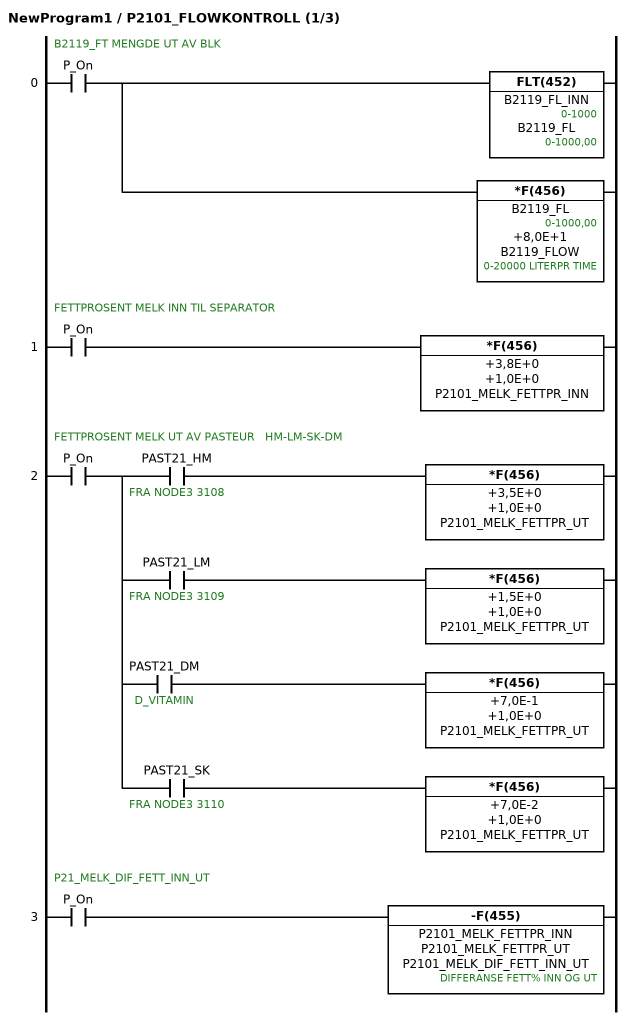
; [picture p1056: NewProgram1 / P2101_FLOWKONTROLL, rungs 0-3]
; rung 0: B2119_FT MENGDE UT AV BLK
LD P_On
FLT(452) B2119_FL_INN B2119_FL  ; 0-1000, 0-1000,00
*F(456) B2119_FL +8,0E+1 B2119_FLOW  ; 0-1000,00, 0-20000 LITERPR TIME
; rung 1: FETTPROSENT MELK INN TIL SEPARATOR
LD P_On
*F(456) +3,8E+0 +1,0E+0 P2101_MELK_FETTPR_INN
; rung 2: FETTPROSENT MELK UT AV PASTEUR   HM-LM-SK-DM
LD P_On
OUT TR0
AND PAST21_HM  ; FRA NODE3 3108
*F(456) +3,5E+0 +1,0E+0 P2101_MELK_FETTPR_UT
LD TR0
AND PAST21_LM  ; FRA NODE3 3109
*F(456) +1,5E+0 +1,0E+0 P2101_MELK_FETTPR_UT
LD TR0
AND PAST21_DM  ; D_VITAMIN
*F(456) +7,0E-1 +1,0E+0 P2101_MELK_FETTPR_UT
LD TR0
AND PAST21_SK  ; FRA NODE3 3110
*F(456) +7,0E-2 +1,0E+0 P2101_MELK_FETTPR_UT
; rung 3: P21_MELK_DIF_FETT_INN_UT
LD P_On
-F(455) P2101_MELK_FETTPR_INN P2101_MELK_FETTPR_UT P2101_MELK_DIF_FETT_INN_UT  ; DIFFERANSE FETT% INN OG UT

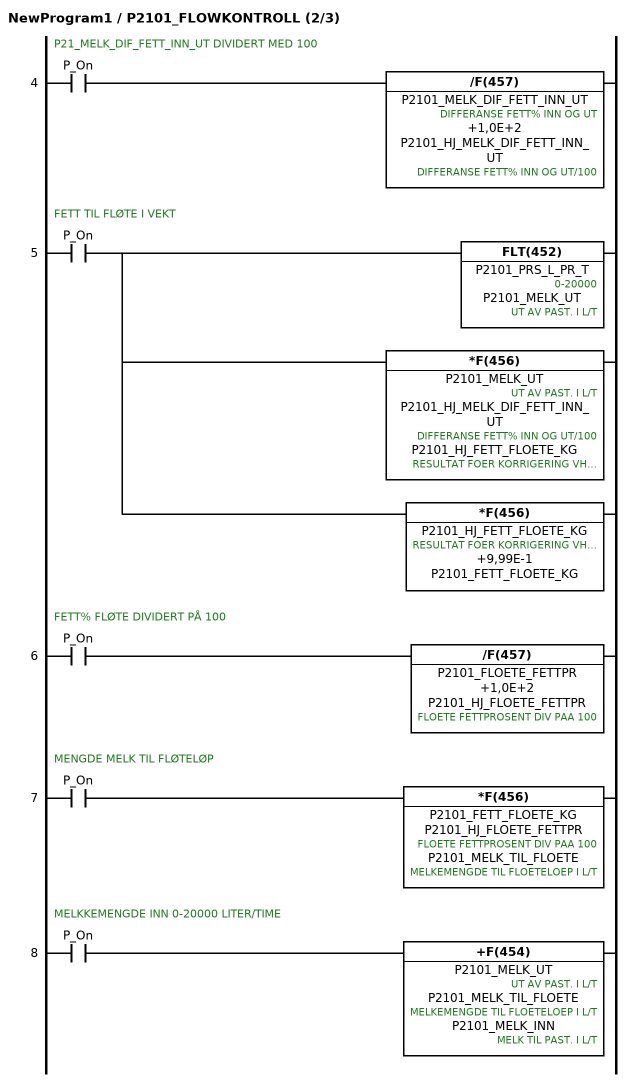
; rung 4: P21_MELK_DIF_FETT_INN_UT DIVIDERT MED 100
LD P_On
/F(457) P2101_MELK_DIF_FETT_INN_UT +1,0E+2 P2101_HJ_MELK_DIF_FETT_INN_UT  ; DIFFERANSE FETT% INN OG UT, DIFFERANSE FETT% INN OG UT/100
; rung 5: FETT TIL FLØTE I VEKT
LD P_On
FLT(452) P2101_PRS_L_PR_T P2101_MELK_UT  ; 0-20000, UT AV PAST. I L/T
*F(456) P2101_MELK_UT P2101_HJ_MELK_DIF_FETT_INN_UT P2101_HJ_FETT_FLOETE_KG  ; UT AV PAST. I L/T, DIFFERANSE FETT% INN OG UT/100, RESULTAT FOER KORRIGERING VHA EGENVEKT
*F(456) P2101_HJ_FETT_FLOETE_KG +9,99E-1 P2101_FETT_FLOETE_KG  ; RESULTAT FOER KORRIGERING VHA EGENVEKT
; rung 6: FETT% FLØTE DIVIDERT PÅ 100
LD P_On
/F(457) P2101_FLOETE_FETTPR +1,0E+2 P2101_HJ_FLOETE_FETTPR  ; FLOETE FETTPROSENT DIV PAA 100
; rung 7: MENGDE MELK TIL FLØTELØP
LD P_On
*F(456) P2101_FETT_FLOETE_KG P2101_HJ_FLOETE_FETTPR P2101_MELK_TIL_FLOETE  ; FLOETE FETTPROSENT DIV PAA 100, MELKEMENGDE TIL FLOETELOEP I L/T
; rung 8: MELKKEMENGDE INN 0-20000 LITER/TIME
LD P_On
+F(454) P2101_MELK_UT P2101_MELK_TIL_FLOETE P2101_MELK_INN  ; UT AV PAST. I L/T, MELKEMENGDE TIL FLOETELOEP I L/T, MELK TIL PAST. I L/T

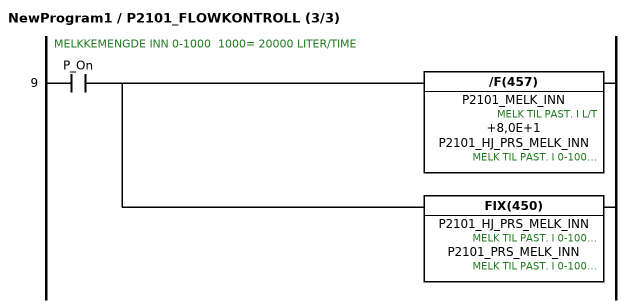
; rung 9: MELKKEMENGDE INN 0-1000  1000= 20000 LITER/TIME
LD P_On
/F(457) P2101_MELK_INN +8,0E+1 P2101_HJ_PRS_MELK_INN  ; MELK TIL PAST. I L/T, MELK TIL PAST. I 0-1000 1000=20000L/T
FIX(450) P2101_HJ_PRS_MELK_INN P2101_PRS_MELK_INN  ; MELK TIL PAST. I 0-1000 1000=20000L/T

### Section P2101

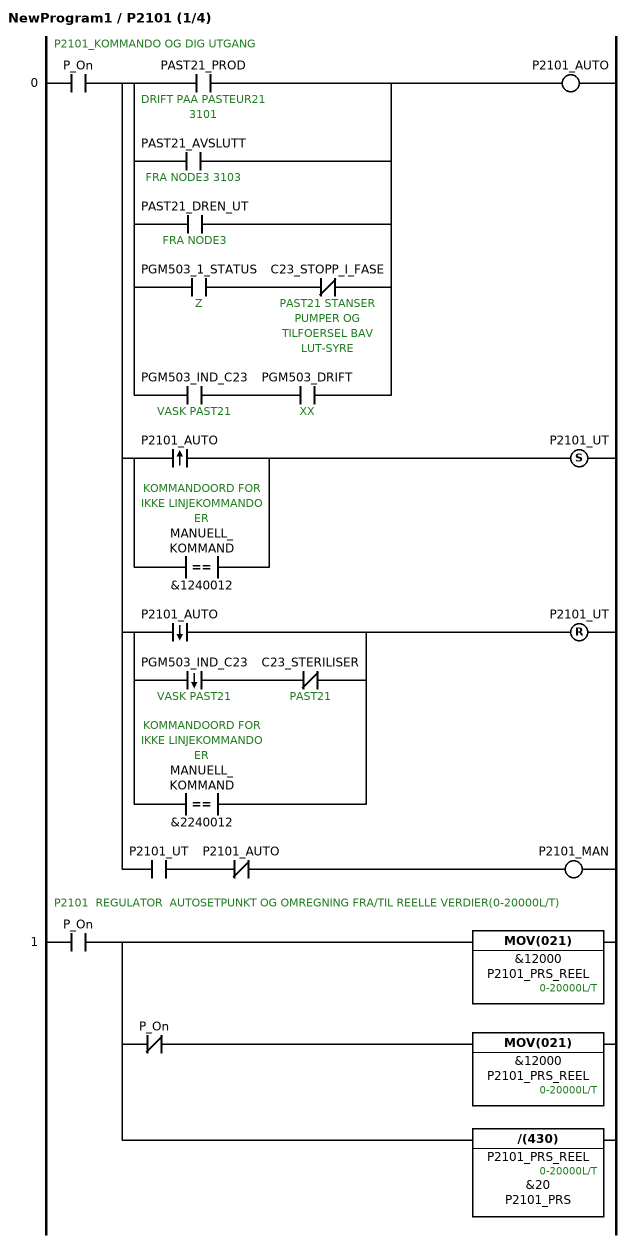
; rung 0: P2101_KOMMANDO OG DIG UTGANG
LD P_On
OUT TR0
LD PAST21_PROD  ; DRIFT PAA PASTEUR21 3101
OR PAST21_AVSLUTT  ; FRA NODE3 3103
OR PAST21_DREN_UT  ; FRA NODE3
LD PGM503_1_STATUS  ; Z
ANDNOT C23_STOPP_I_FASE  ; PAST21 STANSER PUMPER OG TILFOERSEL BAV LUT-SYRE
ORLD
LD PGM503_IND_C23  ; VASK PAST21
AND PGM503_DRIFT  ; XX
ORLD
ANDLD
OUT P2101_AUTO
LD TR0
@LD P2101_AUTO
OR=L(301) MANUELL_KOMMAND &1240012  ; KOMMANDOORD FOR IKKE LINJEKOMMANDOER
ANDLD
SET P2101_UT
LD TR0
%LD P2101_AUTO
%LD PGM503_IND_C23  ; VASK PAST21
ANDNOT C23_STERILISER  ; PAST21
ORLD
OR=L(301) MANUELL_KOMMAND &2240012  ; KOMMANDOORD FOR IKKE LINJEKOMMANDOER
ANDLD
RSET P2101_UT
LD TR0
AND P2101_UT
ANDNOT P2101_AUTO
OUT P2101_MAN
; rung 1: P2101  REGULATOR  AUTOSETPUNKT OG OMREGNING FRA/TIL REELLE VERDIER(0-20000L/T)
LD P_On
OUT TR0
MOV(021) &12000 P2101_PRS_REEL  ; 0-20000L/T
ANDNOT P_On
MOV(021) &12000 P2101_PRS_REEL  ; 0-20000L/T
LD TR0
/(430) P2101_PRS_REEL &20 P2101_PRS  ; 0-20000L/T

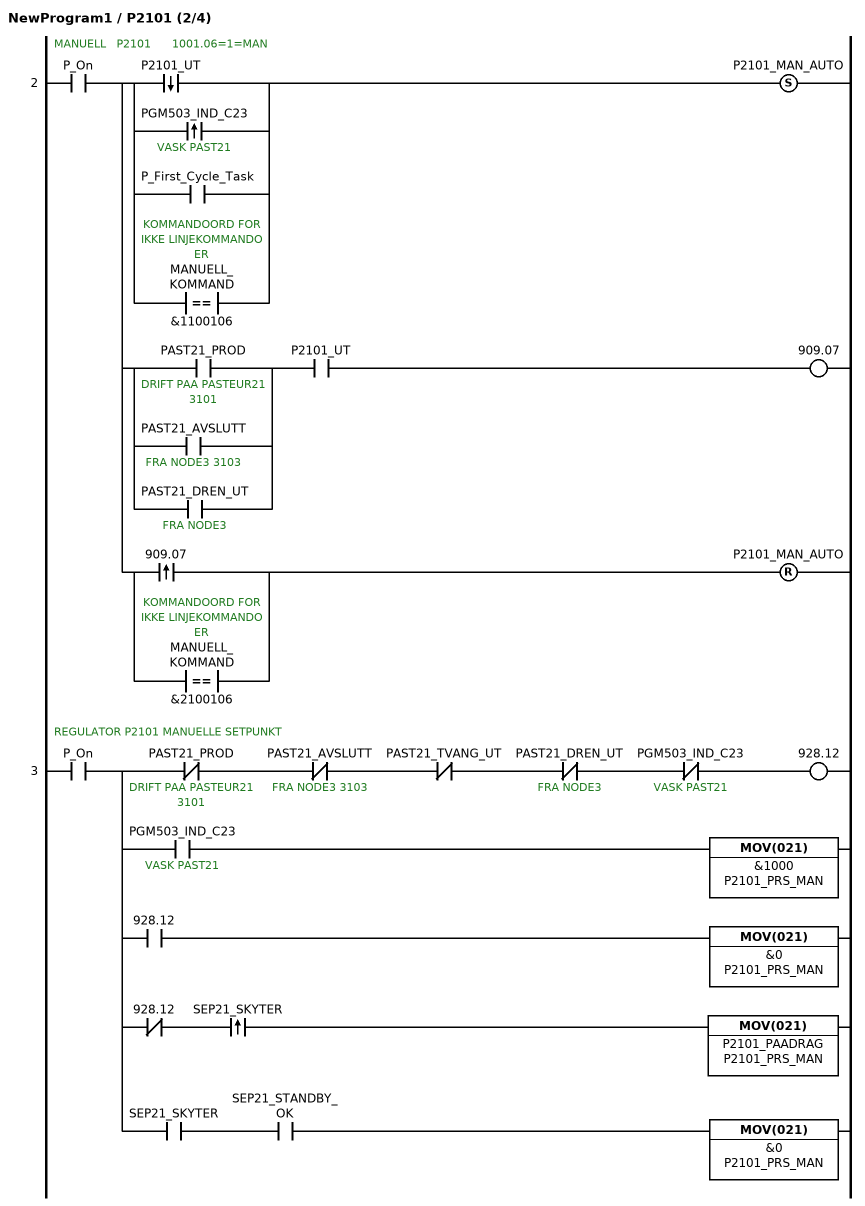
; rung 2: MANUELL   P2101      1001.06=1=MAN
LD P_On
OUT TR0
%LD P2101_UT
@OR PGM503_IND_C23  ; VASK PAST21
OR P_First_Cycle_Task
OR=L(301) MANUELL_KOMMAND &1100106  ; KOMMANDOORD FOR IKKE LINJEKOMMANDOER
ANDLD
SET P2101_MAN_AUTO
LD TR0
LD PAST21_PROD  ; DRIFT PAA PASTEUR21 3101
OR PAST21_AVSLUTT  ; FRA NODE3 3103
OR PAST21_DREN_UT  ; FRA NODE3
ANDLD
AND P2101_UT
OUT 909.07
LD TR0
@LD 909.07
OR=L(301) MANUELL_KOMMAND &2100106  ; KOMMANDOORD FOR IKKE LINJEKOMMANDOER
ANDLD
RSET P2101_MAN_AUTO
; rung 3: REGULATOR P2101 MANUELLE SETPUNKT
LD P_On
OUT TR0
ANDNOT PAST21_PROD  ; DRIFT PAA PASTEUR21 3101
ANDNOT PAST21_AVSLUTT  ; FRA NODE3 3103
ANDNOT PAST21_TVANG_UT
ANDNOT PAST21_DREN_UT  ; FRA NODE3
ANDNOT PGM503_IND_C23  ; VASK PAST21
OUT 928.12
LD TR0
AND PGM503_IND_C23  ; VASK PAST21
MOV(021) &1000 P2101_PRS_MAN
LD TR0
AND 928.12
MOV(021) &0 P2101_PRS_MAN
LD TR0
ANDNOT 928.12
@AND SEP21_SKYTER
MOV(021) P2101_PAADRAG P2101_PRS_MAN
LD TR0
AND SEP21_SKYTER
AND SEP21_STANDBY_OK
MOV(021) &0 P2101_PRS_MAN

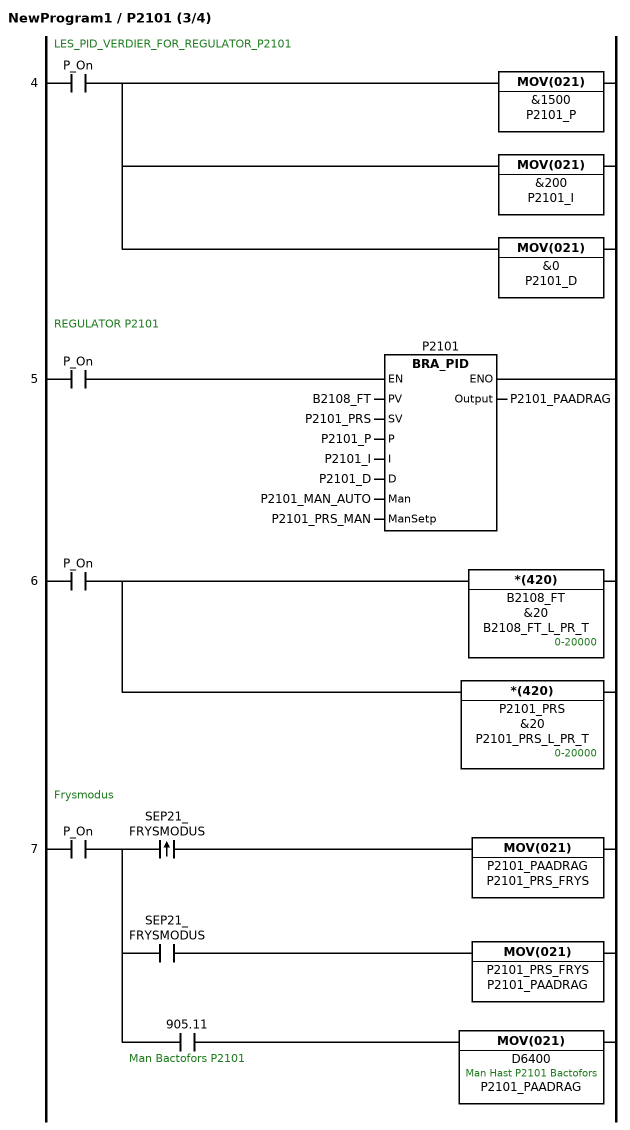
; rung 4: LES_PID_VERDIER_FOR_REGULATOR_P2101
LD P_On
MOV(021) &1500 P2101_P
MOV(021) &200 P2101_I
MOV(021) &0 P2101_D
; rung 5: REGULATOR P2101
LD P_On
CALL P2101 : BRA_PID (PV := B2108_FT, SV := P2101_PRS, P := P2101_P, I := P2101_I, D := P2101_D, Man := P2101_MAN_AUTO, ManSetp := P2101_PRS_MAN, Output => P2101_PAADRAG)
; rung 6
LD P_On
*(420) B2108_FT &20 B2108_FT_L_PR_T  ; 0-20000
*(420) P2101_PRS &20 P2101_PRS_L_PR_T  ; 0-20000
; rung 7: Frysmodus
LD P_On
OUT TR0
@AND SEP21_FRYSMODUS
MOV(021) P2101_PAADRAG P2101_PRS_FRYS
LD TR0
AND SEP21_FRYSMODUS
MOV(021) P2101_PRS_FRYS P2101_PAADRAG
LD TR0
AND 905.11  ; Man Bactofors P2101
MOV(021) D6400 P2101_PAADRAG  ; Man Hast P2101 Bactofors

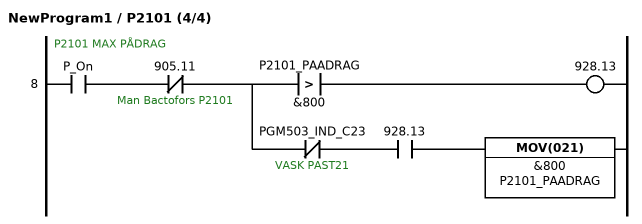
; rung 8: P2101 MAX PÅDRAG
LD P_On
ANDNOT 905.11  ; Man Bactofors P2101
OUT TR0
AND>(320) P2101_PAADRAG &800
OUT 928.13
LD TR0
ANDNOT PGM503_IND_C23  ; VASK PAST21
AND 928.13
MOV(021) &800 P2101_PAADRAG

### Section P2102

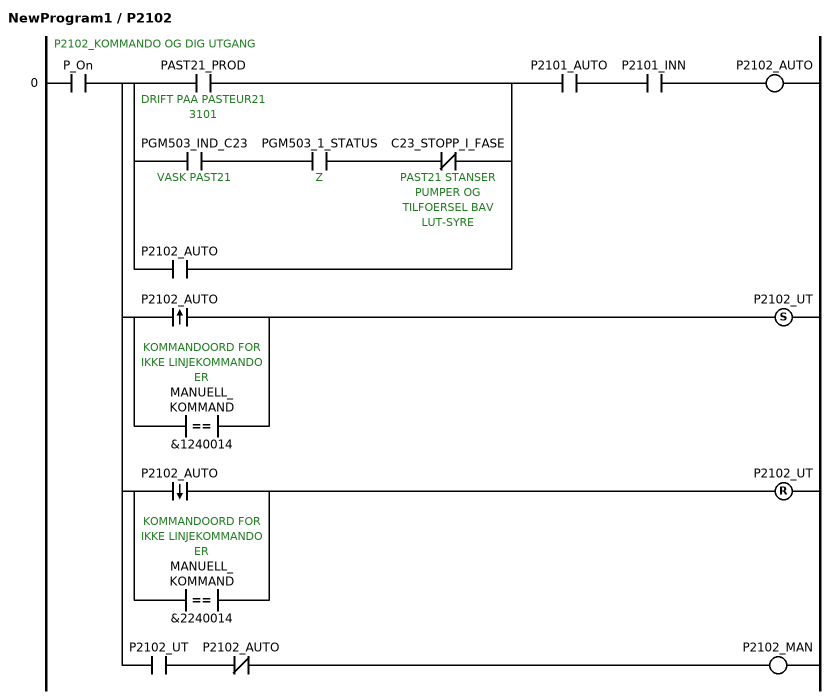
; rung 0: P2102_KOMMANDO OG DIG UTGANG
LD P_On
OUT TR0
LD PAST21_PROD  ; DRIFT PAA PASTEUR21 3101
LD PGM503_IND_C23  ; VASK PAST21
AND PGM503_1_STATUS  ; Z
ANDNOT C23_STOPP_I_FASE  ; PAST21 STANSER PUMPER OG TILFOERSEL BAV LUT-SYRE
ORLD
OR P2102_AUTO
ANDLD
AND P2101_AUTO
AND P2101_INN
OUT P2102_AUTO
LD TR0
@LD P2102_AUTO
OR=L(301) MANUELL_KOMMAND &1240014  ; KOMMANDOORD FOR IKKE LINJEKOMMANDOER
ANDLD
SET P2102_UT
LD TR0
%LD P2102_AUTO
OR=L(301) MANUELL_KOMMAND &2240014  ; KOMMANDOORD FOR IKKE LINJEKOMMANDOER
ANDLD
RSET P2102_UT
LD TR0
AND P2102_UT
ANDNOT P2102_AUTO
OUT P2102_MAN

### Section P2103

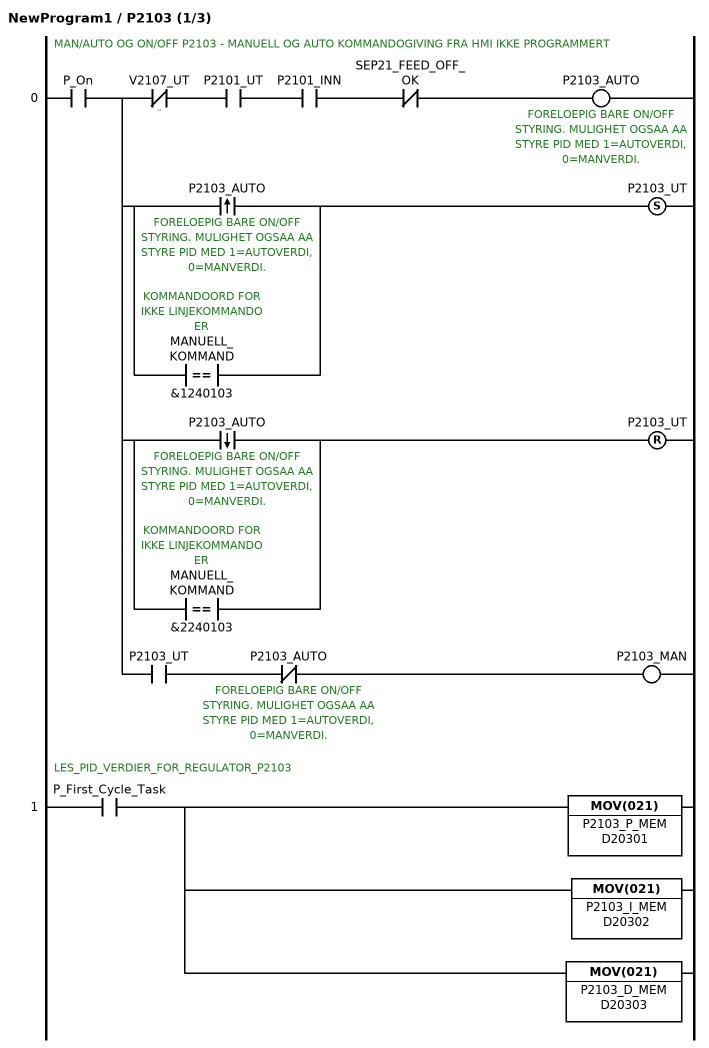
; rung 0: MAN/AUTO OG ON/OFF P2103 - MANUELL OG AUTO KOMMANDOGIVING FRA HMI IKKE PROGRAMMERT
LD P_On
OUT TR0
ANDNOT V2107_UT  ; ¨
AND P2101_UT
AND P2101_INN
ANDNOT SEP21_FEED_OFF_OK
OUT P2103_AUTO  ; FORELOEPIG BARE ON/OFF STYRING. MULIGHET OGSAA AA STYRE PID MED 1=AUTOVERDI, 0=MANVERDI.
LD TR0
@LD P2103_AUTO  ; FORELOEPIG BARE ON/OFF STYRING. MULIGHET OGSAA AA STYRE PID MED 1=AUTOVERDI, 0=MANVERDI.
OR=L(301) MANUELL_KOMMAND &1240103  ; KOMMANDOORD FOR IKKE LINJEKOMMANDOER
ANDLD
SET P2103_UT
LD TR0
%LD P2103_AUTO  ; FORELOEPIG BARE ON/OFF STYRING. MULIGHET OGSAA AA STYRE PID MED 1=AUTOVERDI, 0=MANVERDI.
OR=L(301) MANUELL_KOMMAND &2240103  ; KOMMANDOORD FOR IKKE LINJEKOMMANDOER
ANDLD
RSET P2103_UT
LD TR0
AND P2103_UT
ANDNOT P2103_AUTO  ; FORELOEPIG BARE ON/OFF STYRING. MULIGHET OGSAA AA STYRE PID MED 1=AUTOVERDI, 0=MANVERDI.
OUT P2103_MAN
; rung 1: LES_PID_VERDIER_FOR_REGULATOR_P2103
LD P_First_Cycle_Task
MOV(021) P2103_P_MEM D20301
MOV(021) P2103_I_MEM D20302
MOV(021) P2103_D_MEM D20303

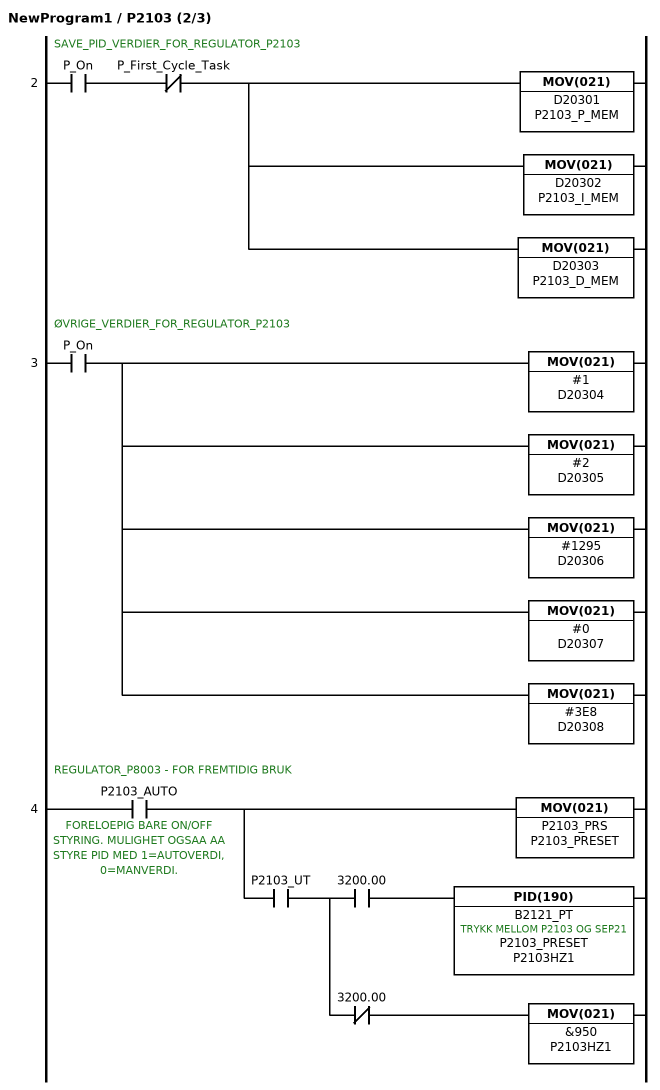
; rung 2: SAVE_PID_VERDIER_FOR_REGULATOR_P2103
LD P_On
ANDNOT P_First_Cycle_Task
MOV(021) D20301 P2103_P_MEM
MOV(021) D20302 P2103_I_MEM
MOV(021) D20303 P2103_D_MEM
; rung 3: ØVRIGE_VERDIER_FOR_REGULATOR_P2103
LD P_On
MOV(021) #1 D20304
MOV(021) #2 D20305
MOV(021) #1295 D20306
MOV(021) #0 D20307
MOV(021) #3E8 D20308
; rung 4: REGULATOR_P8003 - FOR FREMTIDIG BRUK
LD P2103_AUTO  ; FORELOEPIG BARE ON/OFF STYRING. MULIGHET OGSAA AA STYRE PID MED 1=AUTOVERDI, 0=MANVERDI.
MOV(021) P2103_PRS P2103_PRESET
AND P2103_UT
OUT TR0
AND 3200.00
PID(190) B2121_PT P2103_PRESET P2103HZ1  ; TRYKK MELLOM P2103 OG SEP21
LD TR0
ANDNOT 3200.00
MOV(021) &950 P2103HZ1

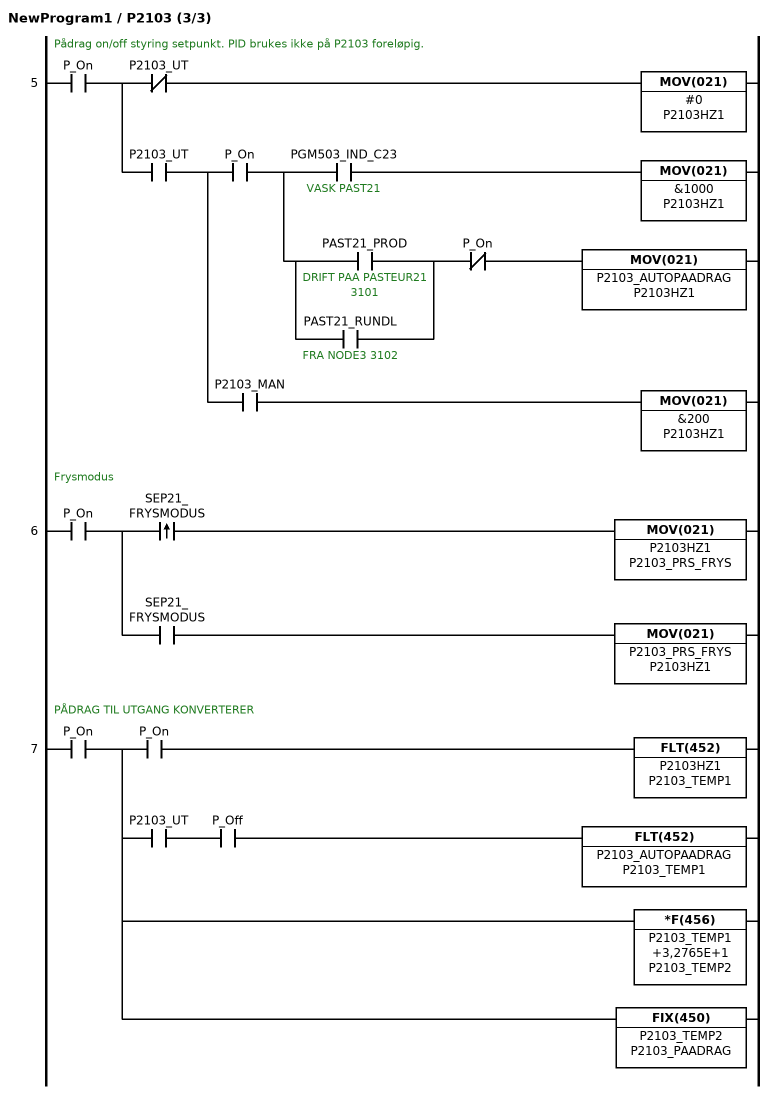
; rung 5: Pådrag on/off styring setpunkt. PID brukes ikke på P2103 foreløpig.
LD P_On
OUT TR0
ANDNOT P2103_UT
MOV(021) #0 P2103HZ1
LD TR0
AND P2103_UT
OUT TR0
AND P_On
OUT TR1
AND PGM503_IND_C23  ; VASK PAST21
MOV(021) &1000 P2103HZ1
LD TR1
LD PAST21_PROD  ; DRIFT PAA PASTEUR21 3101
OR PAST21_RUNDL  ; FRA NODE3 3102
ANDLD
ANDNOT P_On
MOV(021) P2103_AUTOPAADRAG P2103HZ1
LD TR0
AND P2103_MAN
MOV(021) &200 P2103HZ1
; rung 6: Frysmodus
LD P_On
OUT TR0
@AND SEP21_FRYSMODUS
MOV(021) P2103HZ1 P2103_PRS_FRYS
LD TR0
AND SEP21_FRYSMODUS
MOV(021) P2103_PRS_FRYS P2103HZ1
; rung 7: PÅDRAG TIL UTGANG KONVERTERER
LD P_On
OUT TR0
AND P_On
FLT(452) P2103HZ1 P2103_TEMP1  // MAN
LD TR0
AND P2103_UT
AND P_Off
FLT(452) P2103_AUTOPAADRAG P2103_TEMP1  // FRA PID
LD TR0
*F(456) P2103_TEMP1 +3,2765E+1 P2103_TEMP2
FIX(450) P2103_TEMP2 P2103_PAADRAG

### Section P2104

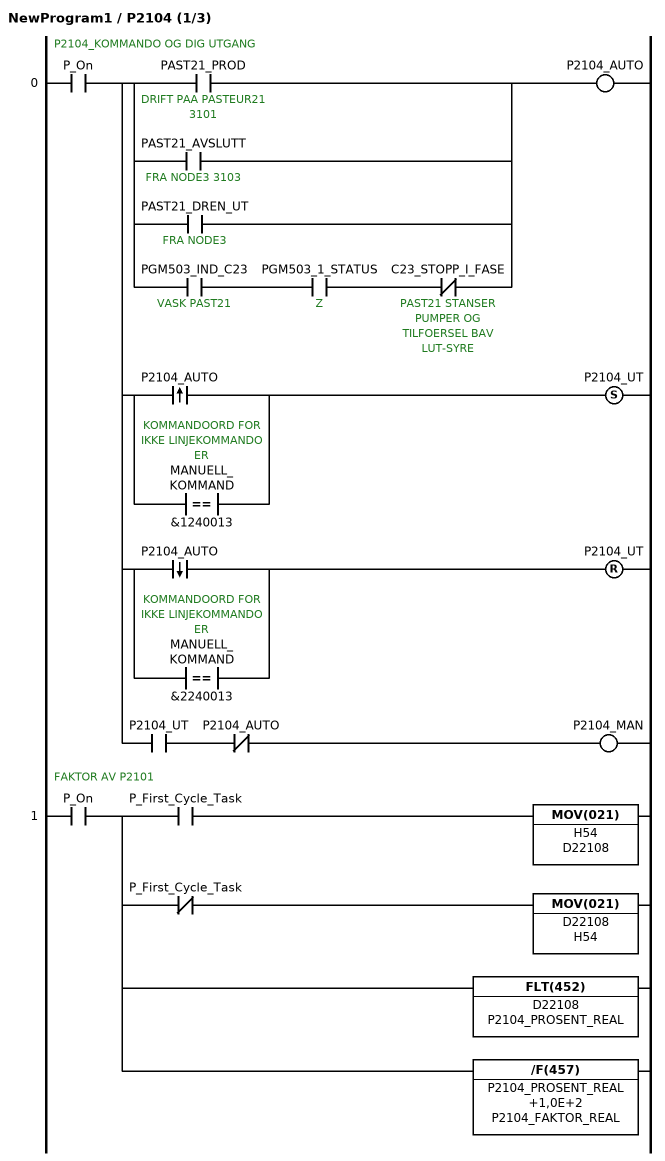
; rung 0: P2104_KOMMANDO OG DIG UTGANG
LD P_On
OUT TR0
LD PAST21_PROD  ; DRIFT PAA PASTEUR21 3101
OR PAST21_AVSLUTT  ; FRA NODE3 3103
OR PAST21_DREN_UT  ; FRA NODE3
LD PGM503_IND_C23  ; VASK PAST21
AND PGM503_1_STATUS  ; Z
ANDNOT C23_STOPP_I_FASE  ; PAST21 STANSER PUMPER OG TILFOERSEL BAV LUT-SYRE
ORLD
ANDLD
OUT P2104_AUTO
LD TR0
@LD P2104_AUTO
OR=L(301) MANUELL_KOMMAND &1240013  ; KOMMANDOORD FOR IKKE LINJEKOMMANDOER
ANDLD
SET P2104_UT
LD TR0
%LD P2104_AUTO
OR=L(301) MANUELL_KOMMAND &2240013  ; KOMMANDOORD FOR IKKE LINJEKOMMANDOER
ANDLD
RSET P2104_UT
LD TR0
AND P2104_UT
ANDNOT P2104_AUTO
OUT P2104_MAN
; rung 1: FAKTOR AV P2101
LD P_On
OUT TR0
AND P_First_Cycle_Task
MOV(021) H54 D22108
LD TR0
ANDNOT P_First_Cycle_Task
MOV(021) D22108 H54
LD TR0
FLT(452) D22108 P2104_PROSENT_REAL
/F(457) P2104_PROSENT_REAL +1,0E+2 P2104_FAKTOR_REAL

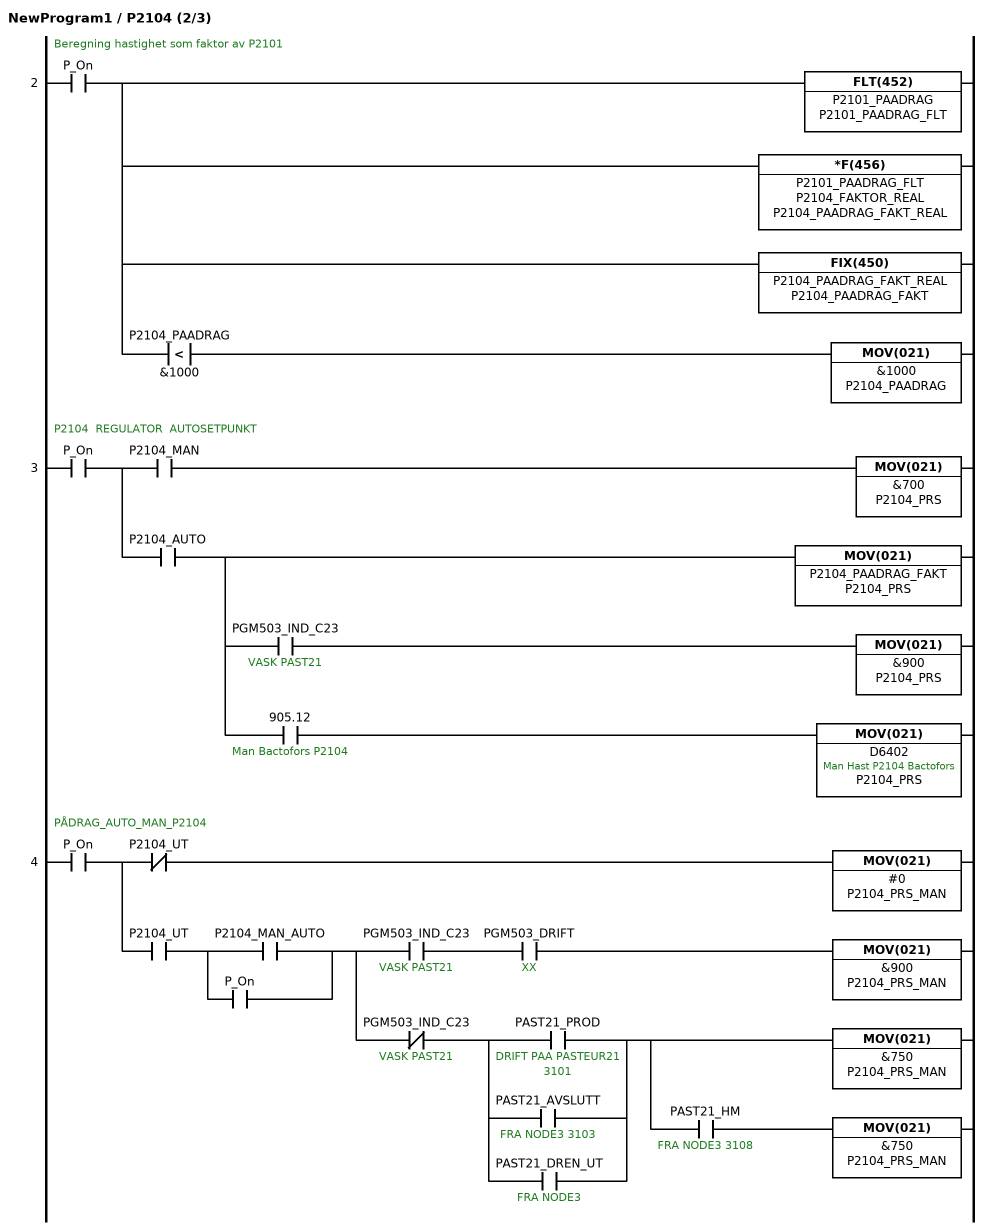
; rung 2: Beregning hastighet som faktor av P2101
LD P_On
FLT(452) P2101_PAADRAG P2101_PAADRAG_FLT
*F(456) P2101_PAADRAG_FLT P2104_FAKTOR_REAL P2104_PAADRAG_FAKT_REAL
FIX(450) P2104_PAADRAG_FAKT_REAL P2104_PAADRAG_FAKT
AND<(310) P2104_PAADRAG &1000
MOV(021) &1000 P2104_PAADRAG
; rung 3: P2104  REGULATOR  AUTOSETPUNKT
LD P_On
OUT TR0
AND P2104_MAN
MOV(021) &700 P2104_PRS
LD TR0
AND P2104_AUTO
OUT TR0
MOV(021) P2104_PAADRAG_FAKT P2104_PRS
AND PGM503_IND_C23  ; VASK PAST21
MOV(021) &900 P2104_PRS
LD TR0
AND 905.12  ; Man Bactofors P2104
MOV(021) D6402 P2104_PRS  ; Man Hast P2104 Bactofors
; rung 4: PÅDRAG_AUTO_MAN_P2104
LD P_On
OUT TR0
ANDNOT P2104_UT
MOV(021) #0 P2104_PRS_MAN
LD TR0
AND P2104_UT
LD P2104_MAN_AUTO
OR P_On
ANDLD
OUT TR0
AND PGM503_IND_C23  ; VASK PAST21
AND PGM503_DRIFT  ; XX
MOV(021) &900 P2104_PRS_MAN
LD TR0
ANDNOT PGM503_IND_C23  ; VASK PAST21
LD PAST21_PROD  ; DRIFT PAA PASTEUR21 3101
OR PAST21_AVSLUTT  ; FRA NODE3 3103
OR PAST21_DREN_UT  ; FRA NODE3
ANDLD
MOV(021) &750 P2104_PRS_MAN
AND PAST21_HM  ; FRA NODE3 3108
MOV(021) &750 P2104_PRS_MAN

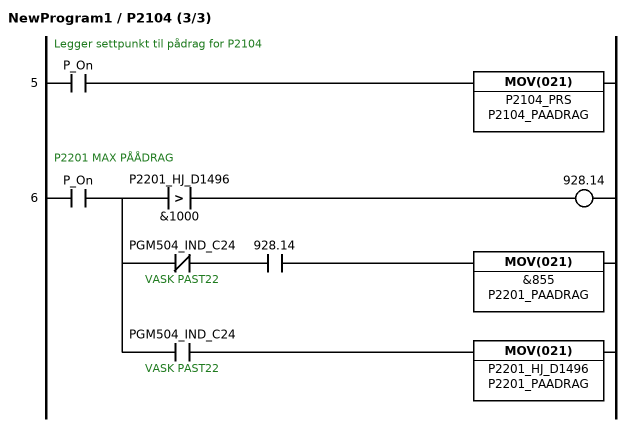
; rung 5: Legger settpunkt til pådrag for P2104
LD P_On
MOV(021) P2104_PRS P2104_PAADRAG
; rung 6: P2201 MAX PÅÅDRAG
LD P_On
OUT TR0
AND>(320) P2201_HJ_D1496 &1000
OUT 928.14
LD TR0
ANDNOT PGM504_IND_C24  ; VASK PAST22
AND 928.14
MOV(021) &855 P2201_PAADRAG
LD TR0
AND PGM504_IND_C24  ; VASK PAST22
MOV(021) P2201_HJ_D1496 P2201_PAADRAG

### Section V2119

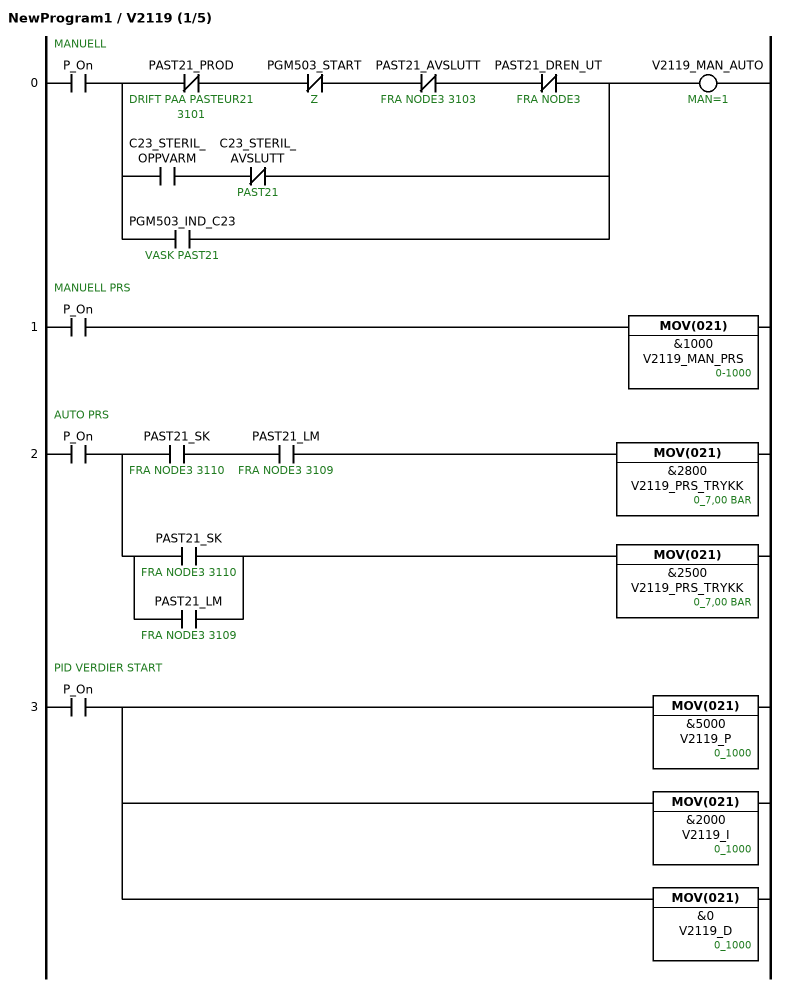
; rung 0: MANUELL
LD P_On
LDNOT PAST21_PROD  ; DRIFT PAA PASTEUR21 3101
ANDNOT PGM503_START  ; Z
ANDNOT PAST21_AVSLUTT  ; FRA NODE3 3103
ANDNOT PAST21_DREN_UT  ; FRA NODE3
LD C23_STERIL_OPPVARM
ANDNOT C23_STERIL_AVSLUTT  ; PAST21
ORLD
OR PGM503_IND_C23  ; VASK PAST21
ANDLD
OUT V2119_MAN_AUTO  ; MAN=1
; rung 1: MANUELL PRS
LD P_On
MOV(021) &1000 V2119_MAN_PRS  ; 0-1000
; rung 2: AUTO PRS
LD P_On
OUT TR0
AND PAST21_SK  ; FRA NODE3 3110
AND PAST21_LM  ; FRA NODE3 3109
MOV(021) &2800 V2119_PRS_TRYKK  ; 0_7,00 BAR
LD TR0
LD PAST21_SK  ; FRA NODE3 3110
OR PAST21_LM  ; FRA NODE3 3109
ANDLD
MOV(021) &2500 V2119_PRS_TRYKK  ; 0_7,00 BAR
; rung 3: PID VERDIER START
LD P_On
MOV(021) &5000 V2119_P  ; 0_1000
MOV(021) &2000 V2119_I  ; 0_1000
MOV(021) &0 V2119_D  ; 0_1000

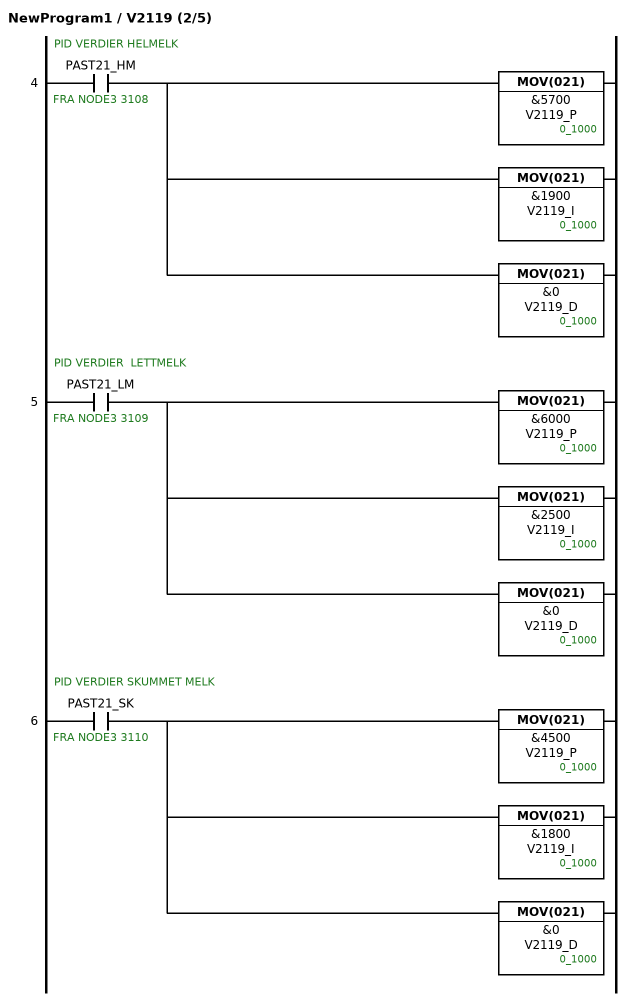
; rung 4: PID VERDIER HELMELK
LD PAST21_HM  ; FRA NODE3 3108
MOV(021) &5700 V2119_P  ; 0_1000
MOV(021) &1900 V2119_I  ; 0_1000
MOV(021) &0 V2119_D  ; 0_1000
; rung 5: PID VERDIER  LETTMELK
LD PAST21_LM  ; FRA NODE3 3109
MOV(021) &6000 V2119_P  ; 0_1000
MOV(021) &2500 V2119_I  ; 0_1000
MOV(021) &0 V2119_D  ; 0_1000
; rung 6: PID VERDIER SKUMMET MELK
LD PAST21_SK  ; FRA NODE3 3110
MOV(021) &4500 V2119_P  ; 0_1000
MOV(021) &1800 V2119_I  ; 0_1000
MOV(021) &0 V2119_D  ; 0_1000

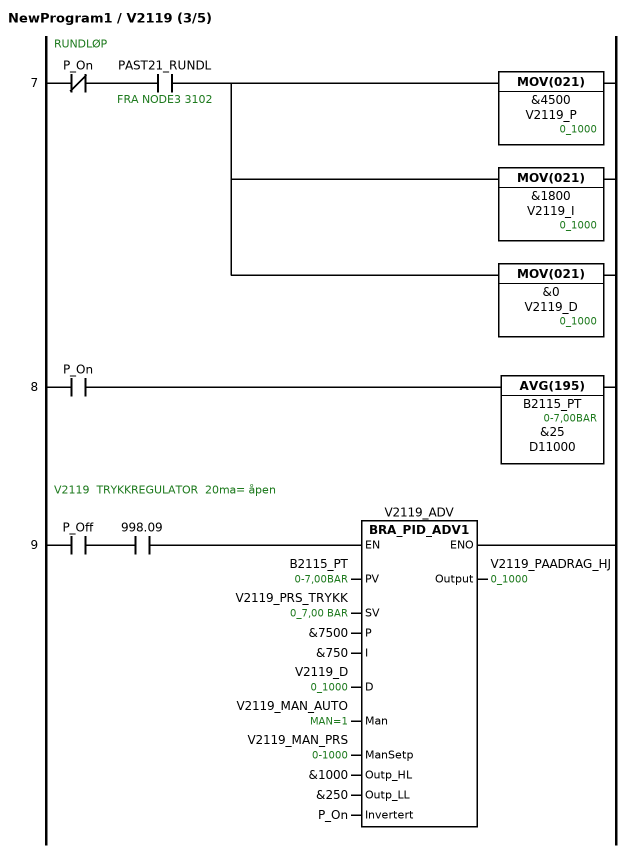
; rung 7: RUNDLØP
LDNOT P_On
AND PAST21_RUNDL  ; FRA NODE3 3102
MOV(021) &4500 V2119_P  ; 0_1000
MOV(021) &1800 V2119_I  ; 0_1000
MOV(021) &0 V2119_D  ; 0_1000
; rung 8
LD P_On
AVG(195) B2115_PT &25 D11000  ; 0-7,00BAR
; rung 9: V2119  TRYKKREGULATOR  20ma= åpen
LD P_Off
AND 998.09
CALL V2119_ADV : BRA_PID_ADV1 (PV := B2115_PT, SV := V2119_PRS_TRYKK, P := &7500, I := &750, D := V2119_D, Man := V2119_MAN_AUTO, ManSetp := V2119_MAN_PRS, Outp_HL := &1000, Outp_LL := &250, Invertert := P_On, Output => V2119_PAADRAG_HJ)  ; 0-7,00BAR, 0_7,00 BAR, 0_1000, MAN=1, 0-1000

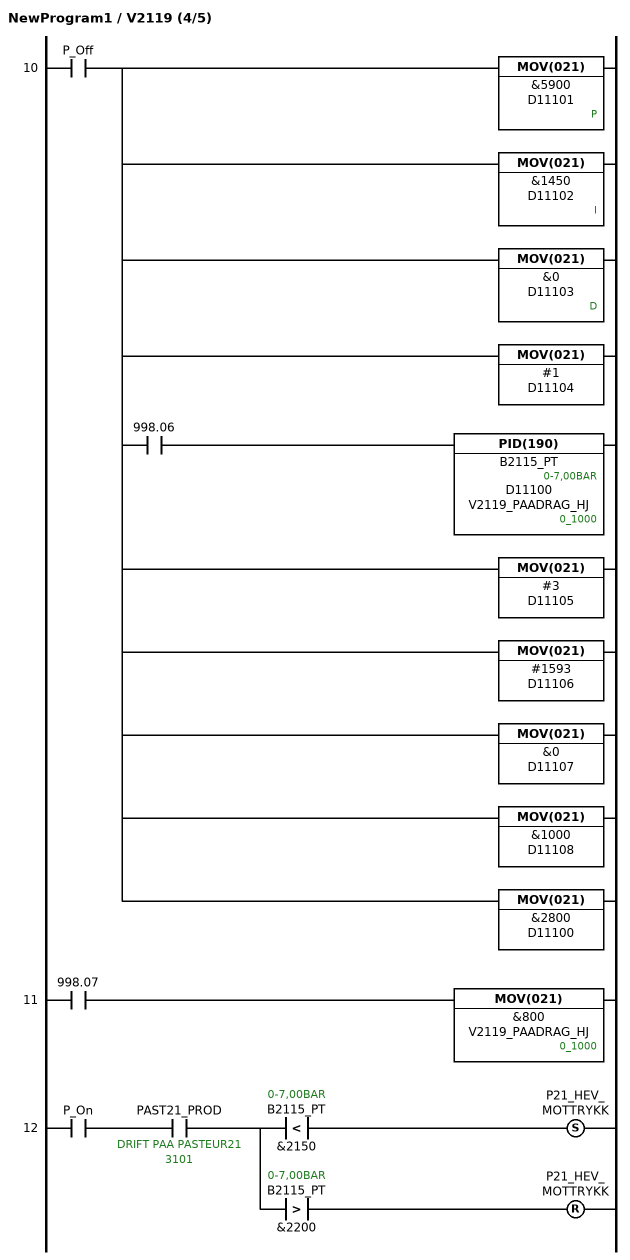
; rung 10
LD P_Off
OUT TR0
MOV(021) &5900 D11101  ; P
MOV(021) &1450 D11102  ; I
MOV(021) &0 D11103  ; D
MOV(021) #1 D11104
AND 998.06
PID(190) B2115_PT D11100 V2119_PAADRAG_HJ  ; 0-7,00BAR, 0_1000
LD TR0
MOV(021) #3 D11105
MOV(021) #1593 D11106
MOV(021) &0 D11107
MOV(021) &1000 D11108
MOV(021) &2800 D11100
; rung 11
LD 998.07
MOV(021) &800 V2119_PAADRAG_HJ  ; 0_1000
; rung 12
LD P_On
AND PAST21_PROD  ; DRIFT PAA PASTEUR21 3101
OUT TR0
AND<(310) B2115_PT &2150  ; 0-7,00BAR
SET P21_HEV_MOTTRYKK
LD TR0
AND>(320) B2115_PT &2200  ; 0-7,00BAR
RSET P21_HEV_MOTTRYKK

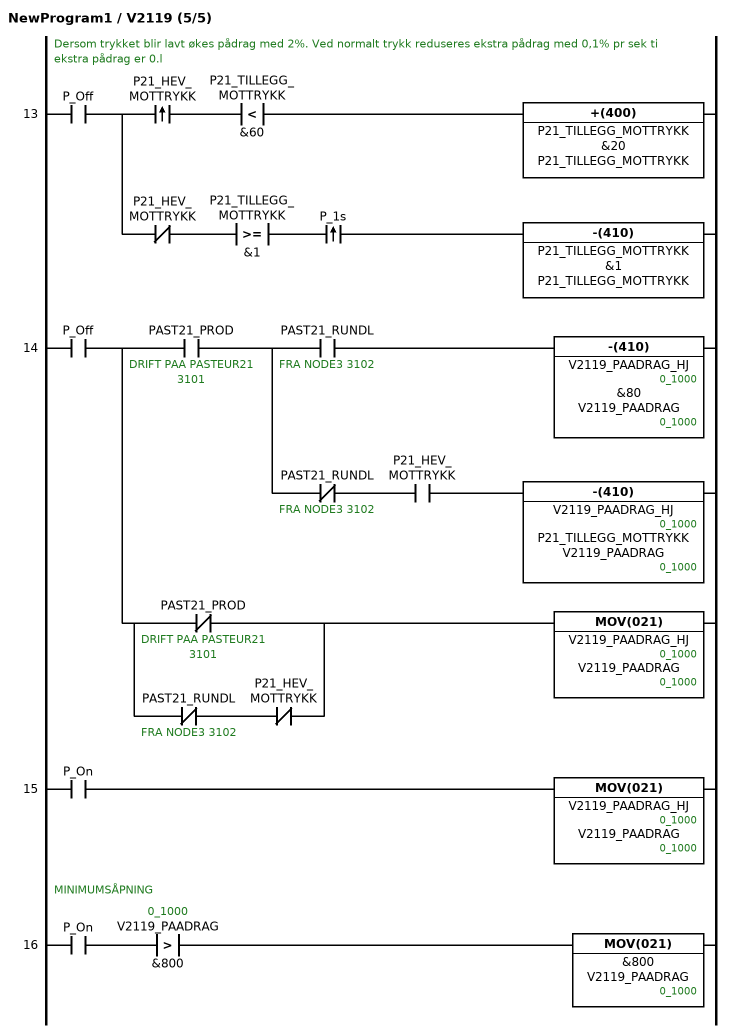
; rung 13: Dersom trykket blir lavt økes pådrag med 2%. Ved normalt trykk reduseres ekstra pådrag med 0,1% pr sek ti ekstra pådrag er 0.l
LD P_Off
OUT TR0
@AND P21_HEV_MOTTRYKK
AND<(310) P21_TILLEGG_MOTTRYKK &60
+(400) P21_TILLEGG_MOTTRYKK &20 P21_TILLEGG_MOTTRYKK
LD TR0
ANDNOT P21_HEV_MOTTRYKK
AND>=(325) P21_TILLEGG_MOTTRYKK &1
@AND P_1s
-(410) P21_TILLEGG_MOTTRYKK &1 P21_TILLEGG_MOTTRYKK
; rung 14
LD P_Off
OUT TR0
AND PAST21_PROD  ; DRIFT PAA PASTEUR21 3101
OUT TR1
AND PAST21_RUNDL  ; FRA NODE3 3102
-(410) V2119_PAADRAG_HJ &80 V2119_PAADRAG  ; 0_1000
LD TR1
ANDNOT PAST21_RUNDL  ; FRA NODE3 3102
AND P21_HEV_MOTTRYKK
-(410) V2119_PAADRAG_HJ P21_TILLEGG_MOTTRYKK V2119_PAADRAG  ; 0_1000
LD TR0
LDNOT PAST21_PROD  ; DRIFT PAA PASTEUR21 3101
LDNOT PAST21_RUNDL  ; FRA NODE3 3102
ANDNOT P21_HEV_MOTTRYKK
ORLD
ANDLD
MOV(021) V2119_PAADRAG_HJ V2119_PAADRAG  ; 0_1000
; rung 15
LD P_On
MOV(021) V2119_PAADRAG_HJ V2119_PAADRAG  ; 0_1000
; rung 16: MINIMUMSÅPNING
LD P_On
AND>(320) V2119_PAADRAG &800  ; 0_1000
MOV(021) &800 V2119_PAADRAG  ; 0_1000

### Section V2161

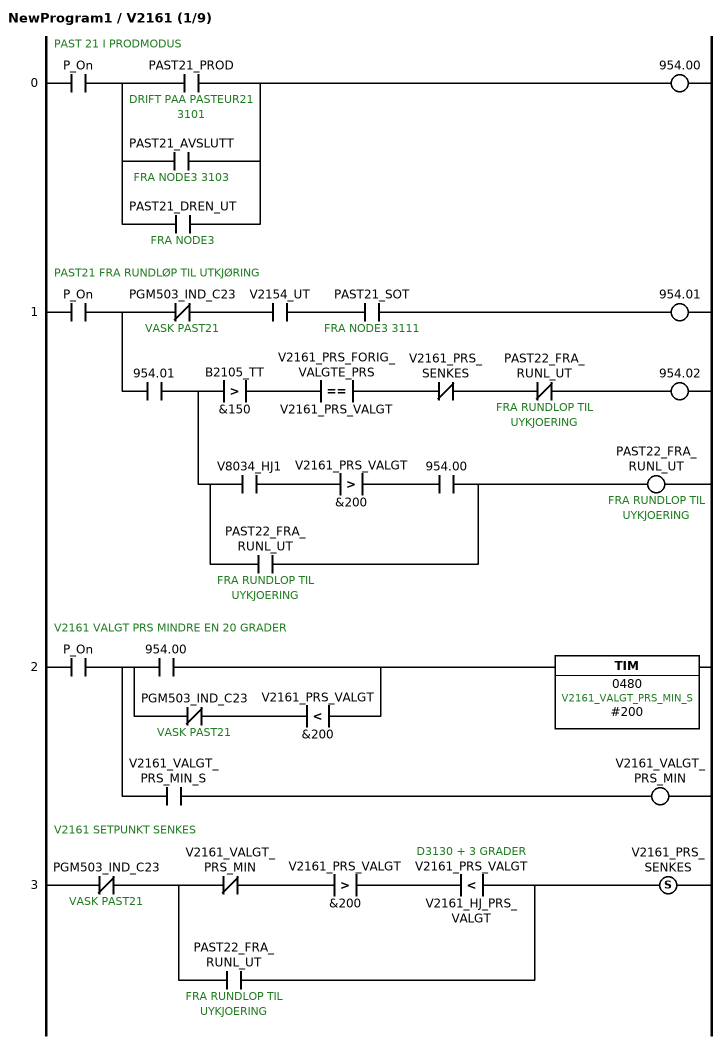
; rung 0: PAST 21 I PRODMODUS
LD P_On
LD PAST21_PROD  ; DRIFT PAA PASTEUR21 3101
OR PAST21_AVSLUTT  ; FRA NODE3 3103
OR PAST21_DREN_UT  ; FRA NODE3
ANDLD
OUT 954.00
; rung 1: PAST21 FRA RUNDLØP TIL UTKJØRING
LD P_On
OUT TR0
ANDNOT PGM503_IND_C23  ; VASK PAST21
AND V2154_UT
AND PAST21_SOT  ; FRA NODE3 3111
OUT 954.01
LD TR0
AND 954.01
OUT TR0
AND>(320) B2105_TT &150
AND=(300) V2161_PRS_FORIG_VALGTE_PRS V2161_PRS_VALGT
ANDNOT V2161_PRS_SENKES
ANDNOT PAST22_FRA_RUNL_UT  ; FRA RUNDLOP TIL UYKJOERING
OUT 954.02
LD TR0
LD V8034_HJ1
AND>(320) V2161_PRS_VALGT &200
AND 954.00
OR PAST22_FRA_RUNL_UT  ; FRA RUNDLOP TIL UYKJOERING
ANDLD
OUT PAST22_FRA_RUNL_UT  ; FRA RUNDLOP TIL UYKJOERING
; rung 2: V2161 VALGT PRS MINDRE EN 20 GRADER
LD P_On
OUT TR0
LD 954.00
LDNOT PGM503_IND_C23  ; VASK PAST21
AND<(310) V2161_PRS_VALGT &200
ORLD
ANDLD
TIM 0480 #200  ; V2161_VALGT_PRS_MIN_S
LD TR0
AND V2161_VALGT_PRS_MIN_S
OUT V2161_VALGT_PRS_MIN
; rung 3: V2161 SETPUNKT SENKES
LDNOT PGM503_IND_C23  ; VASK PAST21
LDNOT V2161_VALGT_PRS_MIN
AND>(320) V2161_PRS_VALGT &200
AND<(310) V2161_PRS_VALGT V2161_HJ_PRS_VALGT  ; D3130 + 3 GRADER
OR PAST22_FRA_RUNL_UT  ; FRA RUNDLOP TIL UYKJOERING
ANDLD
SET V2161_PRS_SENKES

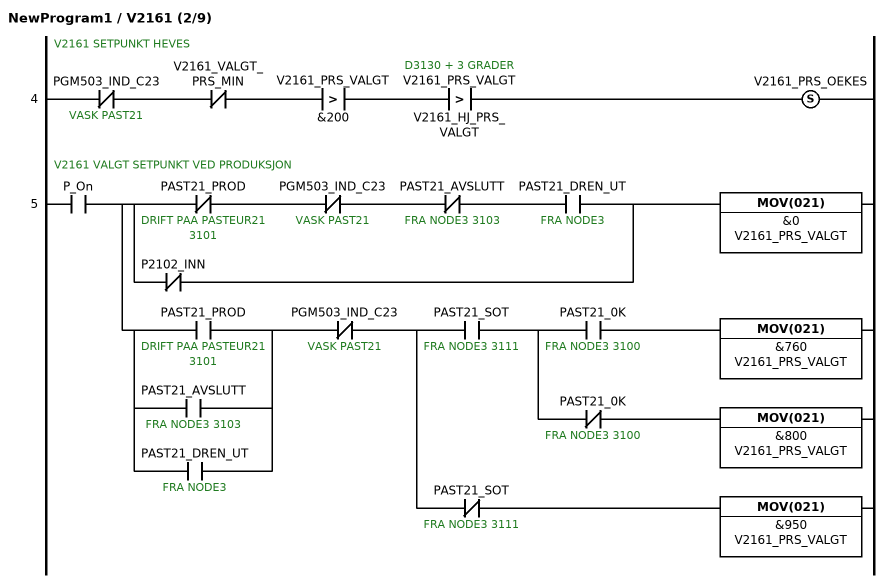
; rung 4: V2161 SETPUNKT HEVES
LDNOT PGM503_IND_C23  ; VASK PAST21
ANDNOT V2161_VALGT_PRS_MIN
AND>(320) V2161_PRS_VALGT &200
AND>(320) V2161_PRS_VALGT V2161_HJ_PRS_VALGT  ; D3130 + 3 GRADER
SET V2161_PRS_OEKES
; rung 5: V2161 VALGT SETPUNKT VED PRODUKSJON
LD P_On
OUT TR0
LDNOT PAST21_PROD  ; DRIFT PAA PASTEUR21 3101
ANDNOT PGM503_IND_C23  ; VASK PAST21
ANDNOT PAST21_AVSLUTT  ; FRA NODE3 3103
AND PAST21_DREN_UT  ; FRA NODE3
ORNOT P2102_INN
ANDLD
MOV(021) &0 V2161_PRS_VALGT
LD TR0
LD PAST21_PROD  ; DRIFT PAA PASTEUR21 3101
OR PAST21_AVSLUTT  ; FRA NODE3 3103
OR PAST21_DREN_UT  ; FRA NODE3
ANDLD
ANDNOT PGM503_IND_C23  ; VASK PAST21
OUT TR0
AND PAST21_SOT  ; FRA NODE3 3111
OUT TR1
AND PAST21_0K  ; FRA NODE3 3100
MOV(021) &760 V2161_PRS_VALGT
LD TR1
ANDNOT PAST21_0K  ; FRA NODE3 3100
MOV(021) &800 V2161_PRS_VALGT
LD TR0
ANDNOT PAST21_SOT  ; FRA NODE3 3111
MOV(021) &950 V2161_PRS_VALGT

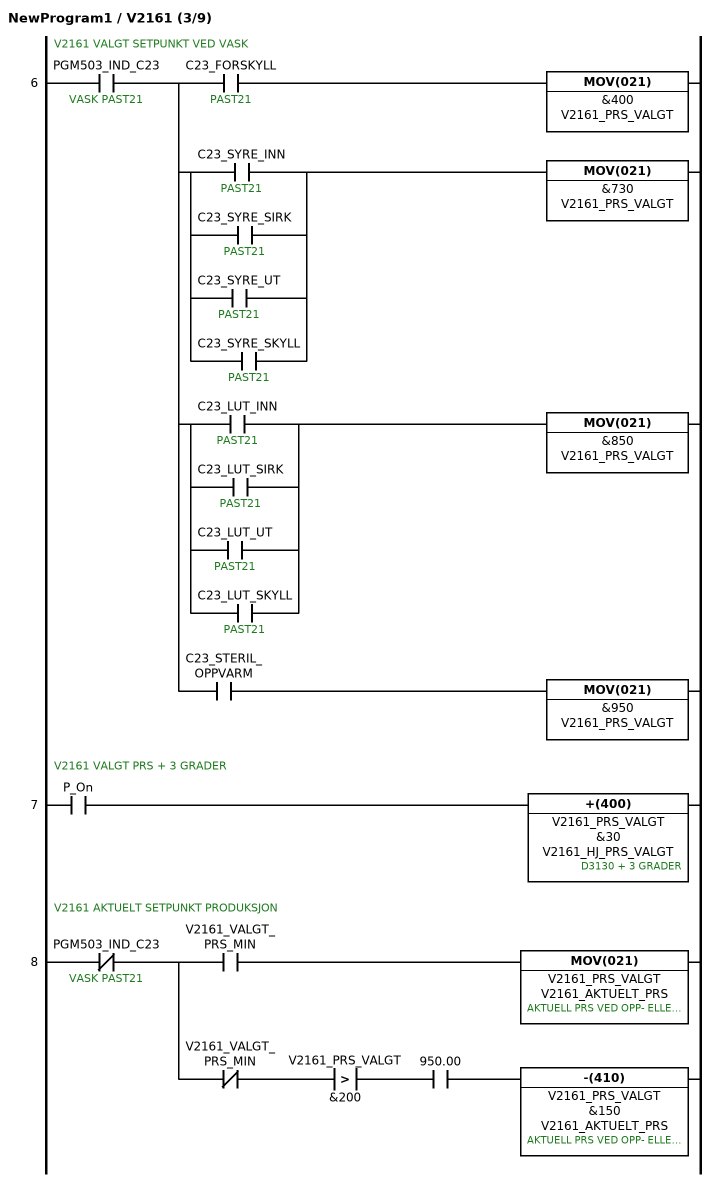
; rung 6: V2161 VALGT SETPUNKT VED VASK
LD PGM503_IND_C23  ; VASK PAST21
OUT TR0
AND C23_FORSKYLL  ; PAST21
MOV(021) &400 V2161_PRS_VALGT
LD TR0
LD C23_SYRE_INN  ; PAST21
OR C23_SYRE_SIRK  ; PAST21
OR C23_SYRE_UT  ; PAST21
OR C23_SYRE_SKYLL  ; PAST21
ANDLD
MOV(021) &730 V2161_PRS_VALGT
LD TR0
LD C23_LUT_INN  ; PAST21
OR C23_LUT_SIRK  ; PAST21
OR C23_LUT_UT  ; PAST21
OR C23_LUT_SKYLL  ; PAST21
ANDLD
MOV(021) &850 V2161_PRS_VALGT
LD TR0
AND C23_STERIL_OPPVARM
MOV(021) &950 V2161_PRS_VALGT
; rung 7: V2161 VALGT PRS + 3 GRADER
LD P_On
+(400) V2161_PRS_VALGT &30 V2161_HJ_PRS_VALGT  ; D3130 + 3 GRADER
; rung 8: V2161 AKTUELT SETPUNKT PRODUKSJON
LDNOT PGM503_IND_C23  ; VASK PAST21
OUT TR0
AND V2161_VALGT_PRS_MIN
MOV(021) V2161_PRS_VALGT V2161_AKTUELT_PRS  ; AKTUELL PRS VED OPP- ELLER NEDTRAPPING
LD TR0
ANDNOT V2161_VALGT_PRS_MIN
AND>(320) V2161_PRS_VALGT &200
AND 950.00
-(410) V2161_PRS_VALGT &150 V2161_AKTUELT_PRS  ; AKTUELL PRS VED OPP- ELLER NEDTRAPPING

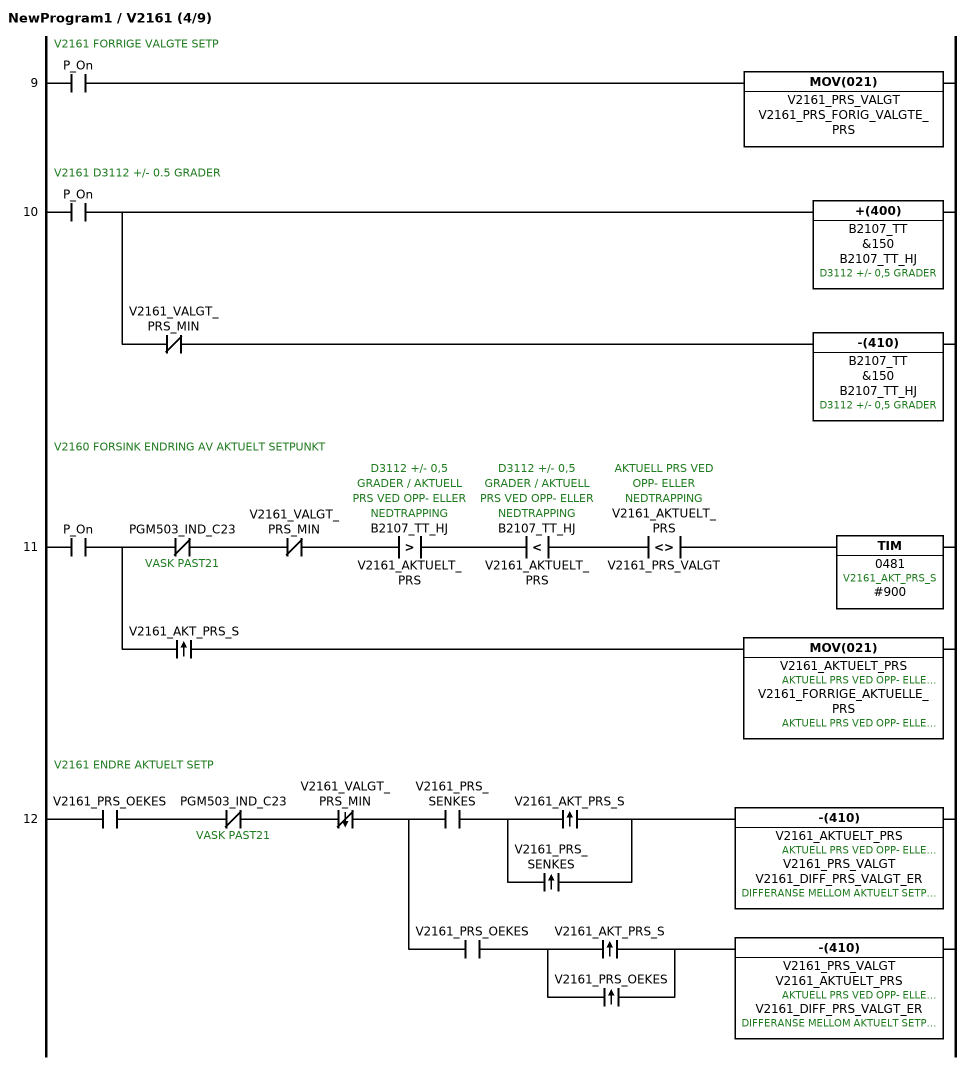
; rung 9: V2161 FORRIGE VALGTE SETP
LD P_On
MOV(021) V2161_PRS_VALGT V2161_PRS_FORIG_VALGTE_PRS
; rung 10: V2161 D3112 +/- 0.5 GRADER
LD P_On
+(400) B2107_TT &150 B2107_TT_HJ  ; D3112 +/- 0,5 GRADER
ANDNOT V2161_VALGT_PRS_MIN
-(410) B2107_TT &150 B2107_TT_HJ  ; D3112 +/- 0,5 GRADER
; rung 11: V2160 FORSINK ENDRING AV AKTUELT SETPUNKT
LD P_On
OUT TR0
ANDNOT PGM503_IND_C23  ; VASK PAST21
ANDNOT V2161_VALGT_PRS_MIN
AND>(320) B2107_TT_HJ V2161_AKTUELT_PRS  ; D3112 +/- 0,5 GRADER, AKTUELL PRS VED OPP- ELLER NEDTRAPPING
AND<(310) B2107_TT_HJ V2161_AKTUELT_PRS  ; D3112 +/- 0,5 GRADER, AKTUELL PRS VED OPP- ELLER NEDTRAPPING
AND<>(305) V2161_AKTUELT_PRS V2161_PRS_VALGT  ; AKTUELL PRS VED OPP- ELLER NEDTRAPPING
TIM 0481 #900  ; V2161_AKT_PRS_S
LD TR0
@AND V2161_AKT_PRS_S
MOV(021) V2161_AKTUELT_PRS V2161_FORRIGE_AKTUELLE_PRS  ; AKTUELL PRS VED OPP- ELLER NEDTRAPPING
; rung 12: V2161 ENDRE AKTUELT SETP
LD V2161_PRS_OEKES
ANDNOT PGM503_IND_C23  ; VASK PAST21
%ANDNOT V2161_VALGT_PRS_MIN
OUT TR0
AND V2161_PRS_SENKES
@LD V2161_AKT_PRS_S
@OR V2161_PRS_SENKES
ANDLD
-(410) V2161_AKTUELT_PRS V2161_PRS_VALGT V2161_DIFF_PRS_VALGT_ER  ; AKTUELL PRS VED OPP- ELLER NEDTRAPPING, DIFFERANSE MELLOM AKTUELT SETP. OG VALGT SETP
LD TR0
AND V2161_PRS_OEKES
@LD V2161_AKT_PRS_S
@OR V2161_PRS_OEKES
ANDLD
-(410) V2161_PRS_VALGT V2161_AKTUELT_PRS V2161_DIFF_PRS_VALGT_ER  ; AKTUELL PRS VED OPP- ELLER NEDTRAPPING, DIFFERANSE MELLOM AKTUELT SETP. OG VALGT SETP

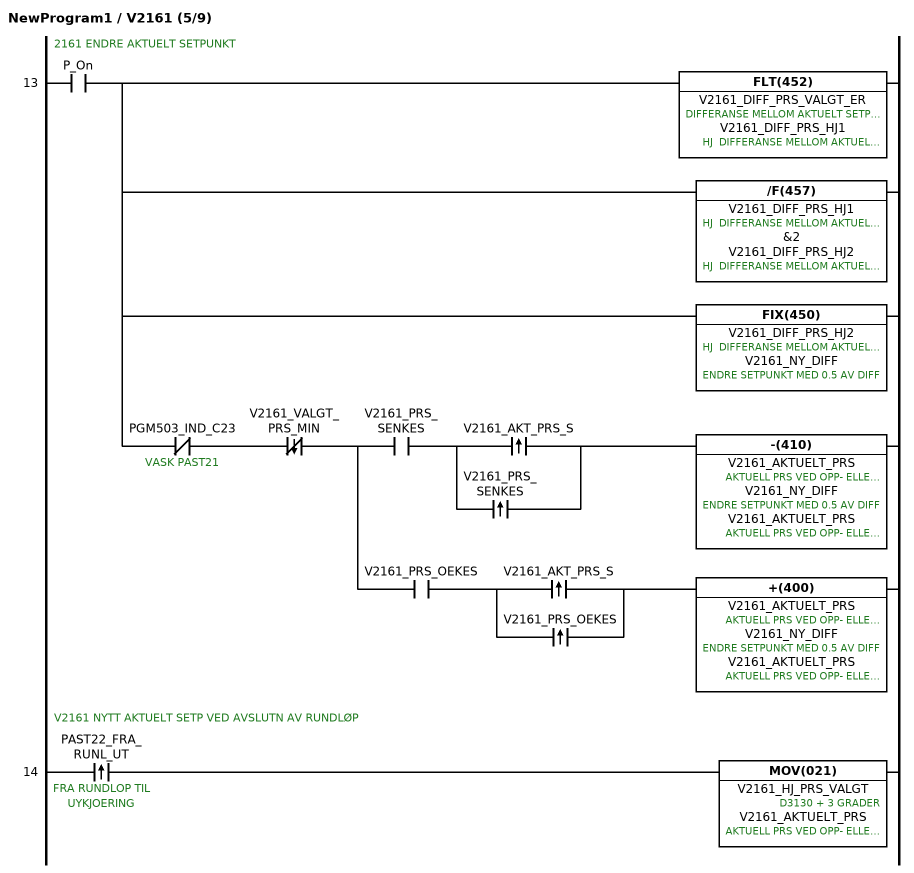
; rung 13: 2161 ENDRE AKTUELT SETPUNKT
LD P_On
FLT(452) V2161_DIFF_PRS_VALGT_ER V2161_DIFF_PRS_HJ1  ; DIFFERANSE MELLOM AKTUELT SETP. OG VALGT SETP, HJ  DIFFERANSE MELLOM AKTUELT SETP. OG VALGT SETP
/F(457) V2161_DIFF_PRS_HJ1 &2 V2161_DIFF_PRS_HJ2  ; HJ  DIFFERANSE MELLOM AKTUELT SETP. OG VALGT SETP
FIX(450) V2161_DIFF_PRS_HJ2 V2161_NY_DIFF  ; HJ  DIFFERANSE MELLOM AKTUELT SETP. OG VALGT SETP, ENDRE SETPUNKT MED 0.5 AV DIFF
ANDNOT PGM503_IND_C23  ; VASK PAST21
%ANDNOT V2161_VALGT_PRS_MIN
OUT TR0
AND V2161_PRS_SENKES
@LD V2161_AKT_PRS_S
@OR V2161_PRS_SENKES
ANDLD
-(410) V2161_AKTUELT_PRS V2161_NY_DIFF V2161_AKTUELT_PRS  ; AKTUELL PRS VED OPP- ELLER NEDTRAPPING, ENDRE SETPUNKT MED 0.5 AV DIFF
LD TR0
AND V2161_PRS_OEKES
@LD V2161_AKT_PRS_S
@OR V2161_PRS_OEKES
ANDLD
+(400) V2161_AKTUELT_PRS V2161_NY_DIFF V2161_AKTUELT_PRS  ; AKTUELL PRS VED OPP- ELLER NEDTRAPPING, ENDRE SETPUNKT MED 0.5 AV DIFF
; rung 14: V2161 NYTT AKTUELT SETP VED AVSLUTN AV RUNDLØP
@LD PAST22_FRA_RUNL_UT  ; FRA RUNDLOP TIL UYKJOERING
MOV(021) V2161_HJ_PRS_VALGT V2161_AKTUELT_PRS  ; D3130 + 3 GRADER, AKTUELL PRS VED OPP- ELLER NEDTRAPPING

